{attribute 'linkalways'} 
{attribute 'no_explicit_call' := 'This FB is a CLASS and must be accessed using methods or properties'}
{attribute 'enable_dynamic_creation'}
FUNCTION_BLOCK FINAL EQ_DWORD EXTENDS Node
VAR
	in1 : _DWORD(0);
	in2 : _DWORD(0);
	out : _BOOL(FALSE);
END_VAR

METHOD PUBLIC Clone : I_Node
VAR
	pNode : POINTER TO EQ_DWORD;
END_VAR
pNode := __NEW(EQ_DWORD);
Clone := pNode^;
END_METHOD

METHOD FB_init : BOOL
VAR_INPUT
	bInitRetains : BOOL; // if TRUE, the retain variables are initialized (warm start / cold start)
	bInCopyCode : BOOL;  // if TRUE, the instance afterwards gets moved into the copy code (online change)
END_VAR
AddInput('in1',THIS^.in1);
AddInput('in2',THIS^.in2);
AddOutput('out', THIS^.out);
END_METHOD

METHOD PROTECTED OnExecute
VAR
END_VAR
out.Value := in1.Value = in2.Value;
END_METHOD

END_FUNCTION_BLOCK

(* stored: Version 1.1.0.1, ProductVersion 3.1.4024.15
   POU EQ_DWORD: Id {d64777cb-223c-44ae-ae70-49b6acc678fd}, SpecialFunc None
   Folder Constructor: Id {af7adf94-545f-44d1-a392-f94a73fad03b}
   Method Clone: Id {d2ddd3b2-02e1-426c-82fe-b4ccabafd1ab}
   Method FB_init: Id {8b76d74b-1353-43b1-89eb-eb1145202160}
   Method OnExecute: Id {d5c83c75-c875-41fa-a506-6d8b1b66ba77} *)
